// TIA Portal project "Parking Garage Indicator" (V17)
// When all parking spots are occupied, a full indicator should turn ON and also barrier should not lift. If the parking spot is vacant, then buzzer will turn ON and barrier will be lifted for 5 sec.

(* hardware
DEVICE "S7-1200 station_1"  S7-1200 Station
   slot 0: "Rack_0"  S7-1200 Rack  Rack  V1.0
   slot 1: "PLC_1"  CPU 1214C AC/DC/Rly  6ES7 214-1BG40-0XB0  V4.5
*)

// ===== PLC "PLC_1"  CPU 1214C AC/DC/Rly =====

VAR_GLOBAL   // PLC tag table "Default tag table"
   "sensor_1" AT %I0.0 : Bool;
   "sensor_2" AT %I0.1 : Bool;
   "sensor_3" AT %I0.2 : Bool;
   "sensor_4" AT %I0.3 : Bool;
   "Full_Indicator" AT %Q0.0 : Bool;
   "Barrier" AT %Q0.1 : Bool;
   "Entrance_Vehicle_Sensor" AT %I0.4 : Bool;
   "Buzzer" AT %Q0.2 : Bool;
END_VAR

// folder: System blocks/Program resources

DATA_BLOCK "IEC_Timer_0_DB"   // DB1
{ S7_Optimized_Access := 'TRUE' }
AUTHOR : Simatic
FAMILY : IEC
NAME : IEC_TMR
VERSION : 1.0
// stored: InstanceOfName IEC_TIMER
"IEC_TIMER"
BEGIN
END_DATA_BLOCK

// folder: (top level)

ORGANIZATION_BLOCK "Main"   // OB1, LAD, ProgramCycle
TITLE = "Main Program Sweep (Cycle)"
{ S7_Optimized_Access := 'TRUE' }
VERSION : 0.1
// Condition: When all sensors are high, meaning all spaces are occupied and no more parking space is leftout for new vehicle, then Full-Indicator light glows.
   VAR_INPUT
      Initial_Call : Bool;   // Initial call of this OB
      Remanence : Bool;   // =True, if remanent data are available
   END_VAR
BEGIN

REGION Network 1
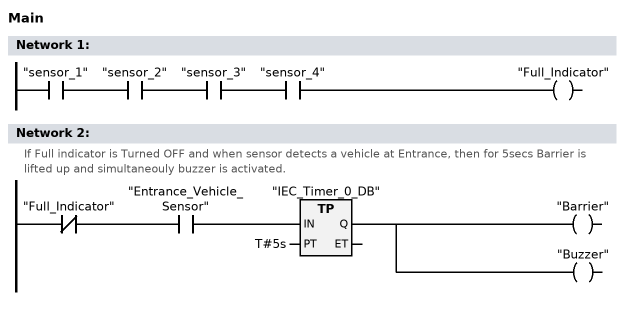
   RUNG wire#powerrail
      Contact( "sensor_1" )
      Contact( "sensor_2" )
      Contact( "sensor_3" )
      Contact( "sensor_4" )
      Coil( "Full_Indicator" )
   END_RUNG
   // the same network as SCL:
   "Full_Indicator" := "sensor_1" AND "sensor_2" AND "sensor_3" AND "sensor_4";
END_REGION

REGION Network 2
   // If Full indicator is Turned OFF and when sensor detects a vehicle at Entrance, then for 5secs Barrier is lifted up and simultaneouly buzzer is activated.
   "IEC_Timer_0_DB".TP(IN := NOT "Full_Indicator" AND "Entrance_Vehicle_Sensor", PT := T#5s);
   "Barrier" := "IEC_Timer_0_DB".Q;
   "Buzzer" := "IEC_Timer_0_DB".Q;
END_REGION
END_ORGANIZATION_BLOCK